Fanuc KAREL source: ORIENT.kl

PROGRAM T
%NOLOCKGROUP
VAR
 v0 : POSITION
 res : VECTOR
BEGIN
 res = ORIENT(v0)
END T
